INTERFACE ITF_ITC EXTENDS __System.IQueryInterface

METHOD M_AddData : BOOL
VAR_INPUT
	meChannelSrc	: E_MFCS_Channel;
	mMsgType		: INT;
	mpData			: PVOID;
	mLen			: UDINT;
END_VAR
END_METHOD

METHOD M_CallITC_Service : BOOL
VAR_INPUT
END_VAR
END_METHOD

METHOD M_Init : BOOL
(**************************************************************************************
 * 	Application		:	BoxControl Framework
 *	Revision		:	$Revision: 355272 $
 *	Revision date	:	$Date: 2015-09-23 11:26:06 +0200 (Wed, 23 Sep 2015) $
 *	Last changed by	:	$Author: b7bolm $
 *	URL				:	$URL: http://almscdc.swisslog.com/repo/SWPD/Development/BoxControlFramework/20_Release/trunk/01_Software/BoxControlFramework/BoxControlFramework/JumpStart/11_Library/10_Application/11_Communication/12_MFCS/11_SIS/11_SIS_6_0/FB_SIS_MsgManager_6_0.TcPOU $
 *
 *	Purpose			:	Initialize 
 *
 * ------------------------------------------------------------------------------------
 *	Copyright Swisslog [IP AG], Switzerland. All rights reserved.
 * 
 * ------------------------------------------------------------------------------------
 *	
 * 	Revision History: 
 *
 * 	VERSION			DATE			INITIALS			DESCRIPTION
 *	0.1				01.01.2001		swl					Example
 *
 **************************************************************************************)
VAR_INPUT
	mInit		: BOOL; // Force init
END_VAR
END_METHOD

METHOD M_SendData : BOOL
VAR_INPUT
	meChannel	: E_MFCS_Channel;
	mMsgType	: INT;
	mpData		: PVOID;
	mLen		: UDINT;
END_VAR
END_METHOD

END_INTERFACE

(* stored: Version 1.1.0.1, ProductVersion 3.1.4022.12
   Itf ITF_ITC: Id {4e81ac09-73f0-4416-bde9-20732eb16d3c}
   Method M_AddData: Id {bc4e74ec-762e-41b8-a1ad-97807f292370}
   Method M_CallITC_Service: Id {e8987561-afe4-47da-95aa-f60605713def}
   Method M_Init: Id {1fbdae60-bb85-4bc1-a544-149ac483c0b9}
   Method M_SendData: Id {55b5b8bb-81f2-4a07-b722-77cc4ff83045} *)
